// TwinCAT 3 PLC project Main
// ProgramVersion: 3.1.4023.0
// libraries:
//   mobject-core, * (mobject.io)
//   Tc2_Standard, * (Beckhoff Automation GmbH)
//   Tc2_System, * (Beckhoff Automation GmbH)
//   Tc3_Module, * (Beckhoff Automation GmbH)
// project tree:
//   / PlcTask.TcTTO
//   POUs/CommandExamples/Cylinder/Commands/ Cylinder_ExtendCommand.TcPOU
//   POUs/CommandExamples/Cylinder/ I_Cylinder.TcIO (not stored), SimulationTwoPositionCylinderWithFeedback.TcPOU
//   POUs/CyclicInstanceExamples/ ExampleFlashingLamp_Composition.TcPOU, ExampleFlashingLamp_Inheritance.TcPOU
//   POUs/ Main.TcPOU
// real-time tasks:
//   TASK PlcTask: cycle T#10ms, priority 20, ADS port 350

CONFIGURATION Main
    RESOURCE PLC ON TwinCAT3
        TASK PlcTask(INTERVAL := T#10ms, PRIORITY := 20);
        PROGRAM Main WITH PlcTask : Main;
    END_RESOURCE
END_CONFIGURATION

// ---- POUs/Main.TcPOU
PROGRAM Main
VAR
	
	task : Task;
	
	// currently only objects created in the same POU as the task will be automatically called.  
	// this will be extended in the next version to allow objects from other POUs and GVLs to be marked
	// as being owned by an alternative task. 
	
	// cyclic instance example
	lamp_inheritance : ExampleFlashingLamp_Inheritance;
	lamp_composed : ExampleFlashingLamp_Composition;
	output1, output2 : BOOL;
	
	// asyncCommand example
	cylinder : SimulationTwoPositionCylinderWithFeedback;
	extendCommand : Cylinder_ExtendCommand(cylinder);
	extendCommandFeedback : I_CommandFeedback;
	extendTrigger : BOOL; // set true to execute the async command
	extendComplete :  BOOL; // will set true once the command completes
	
END_VAR

// all mobject code requires a task object to be made in the calling POU, with the CyclicCall being called. 
task.CyclicCall();

// cyclic instance example
// -----------------------
// the outputs below will flash, even though you are not explicitally calling the cyclic update of the lamps.  
// this allows you as the designer to mark your instances as cyclicInstances for them to automatically call.  
// this is especially useful when passing cyclic objects in as a dependency to non-cyclic objects, or if a non-cyclic object
// makes a cyclic object.  You no longer need to worry about how it will be called.  

output1 := lamp_inheritance.Output;
output2 := lamp_composed.Output;

// asyncCommand example
// --------------------
// asynchronous commands are a special  type of cyclicInstance who only automatically cyclic call when executed.  
// They then unregister themselves once the command is no longer busy. 

IF extendTrigger THEN
	extendTrigger := FALSE;
	extendComplete := FALSE;
	// once you call execute, the command will automatically cyclic call until either done or errored. 
	extendCommand.Execute(extendCommandFeedback);
END_IF

// you can monitor the state of the command using the feedback, although this is not a requirement.  
IF extendCommandFeedback <> 0 AND_THEN extendCommandFeedback.Done THEN
	extendComplete := TRUE;
	extendCommandFeedback.Release();
	extendCommandFeedback := 0;
END_IF

END_PROGRAM

// ---- POUs/CyclicInstanceExamples/ExampleFlashingLamp_Inheritance.TcPOU
FUNCTION_BLOCK ExampleFlashingLamp_Inheritance EXTENDS CyclicInstance
VAR
	// these timers are required to implement the flashing lamp object
	tick : ton;
	tock : ton;
END_VAR

//... no code should go here.

METHOD CyclicCall
VAR_INPUT
END_VAR
tick(in:=NOT tock.Q,pt:=T#1S);
tock(in:=tick.Q,pt:=T#1S);
END_METHOD

PROPERTY PUBLIC Output : BOOL
GET
Output := tick.Q;
END_GET
END_PROPERTY

END_FUNCTION_BLOCK

// ---- POUs/CyclicInstanceExamples/ExampleFlashingLamp_Composition.TcPOU
FUNCTION_BLOCK ExampleFlashingLamp_Composition IMPLEMENTS I_CyclicCalled
VAR
	cyclicCall : AutomaticCyclicCall(THIS^);
	tick : ton;
	tock : ton;
END_VAR

// To make an object automatic cyclic called via composition then you must simply implement I_CyclicCalled 
// and instatiate an AutomaticCyclicCall with your object in the constructor.

// Handy Hint!
// -----------
// if you want to be able to switch the cyclic calling on and off then you can use ManualCyclicCall for 
// this with the .Enable() and .Disable() to control the cyclic state.  ManualCyclic call is use inside
// AsynchronousCommand.

METHOD CyclicCall
VAR_INPUT
END_VAR
tick(in:=NOT tock.Q,pt:=T#1S);
tock(in:=tick.Q,pt:=T#1S);
END_METHOD

PROPERTY PUBLIC Output : BOOL
GET
Output := tick.Q;
END_GET
END_PROPERTY

END_FUNCTION_BLOCK

// ---- POUs/CommandExamples/Cylinder/SimulationTwoPositionCylinderWithFeedback.TcPOU
FUNCTION_BLOCK SimulationTwoPositionCylinderWithFeedback EXTENDS CyclicInstance IMPLEMENTS I_Cylinder
VAR
	Output_Extend AT %Q* : BOOL;
	Output_Retract AT %Q* : BOOL;
	Input_Extended AT %I* : BOOL;
	Input_Retracted AT %I* : BOOL;
	retract, extend : TON;
END_VAR

METHOD PUBLIC CyclicCall
VAR_INPUT
END_VAR
retract(IN:=Output_Retract,PT:=T#2S);
extend(IN:=Output_Extend,PT:=T#2S);

Input_Retracted := retract.Q;
Input_Extended := extend.Q;
END_METHOD

METHOD PUBLIC FullyExtend
VAR_INPUT
END_VAR
Output_Extend := TRUE;
Output_Retract := FALSE;
END_METHOD

METHOD PUBLIC FullyRetract
VAR_INPUT
END_VAR
Output_Extend := FALSE;
Output_Retract := TRUE;
END_METHOD

PROPERTY PUBLIC IsExtending : BOOL
GET
IsExtending := (Output_Extend and not IsFullyExtended);
END_GET
END_PROPERTY

PROPERTY PUBLIC IsFullyExtended : BOOL
GET
IsFullyExtended := extend.Q;
END_GET
END_PROPERTY

PROPERTY PUBLIC IsFullyRetracted : BOOL
GET
IsFullyRetracted := retract.Q;
END_GET
END_PROPERTY

PROPERTY PUBLIC IsRetracting : Bool
GET
IsRetracting := (Output_Retract and not IsFullyRetracted);
END_GET
END_PROPERTY

END_FUNCTION_BLOCK

// ---- POUs/CommandExamples/Cylinder/Commands/Cylinder_ExtendCommand.TcPOU
{attribute 'enable_dynamic_creation'}
FUNCTION_BLOCK Cylinder_ExtendCommand EXTENDS Command
VAR
	cylinder : I_Cylinder;
END_VAR

METHOD FB_init : BOOL
VAR_INPUT
	bInitRetains : BOOL; // if TRUE, the retain variables are initialized (warm start / cold start)
	bInCopyCode : BOOL;  // if TRUE, the instance afterwards gets moved into the copy code (online change)	
	Cylinder : I_Cylinder;
END_VAR
THIS^.cylinder := Cylinder;
END_METHOD

METHOD PROTECTED WhileBusy
VAR_INPUT
	commandState : I_CommandBusyState;
END_VAR
cylinder.FullyExtend();

IF cylinder.IsFullyExtended THEN
	commandState.SetDone();	
END_IF
END_METHOD

END_FUNCTION_BLOCK
